// LS Electric XG5000 project: 래더
// PLC NewPLC
// module base 0 slot 0: 입출력 모듈:XBC-DR32H (DC 24V 입력, 릴레이 출력 32점)
// module base 0 slot 1: 위치결정 모듈:XBF-PD02A (위치결정 펄스(LD)출력형, 2축)
// module base 0 slot 2: 출력 모듈:XBE-TN/TP16A (트랜지스터 출력, 16점 (싱크출력/소스출력))

PROGRAM NewProgram (task: 스캔 프로그램)

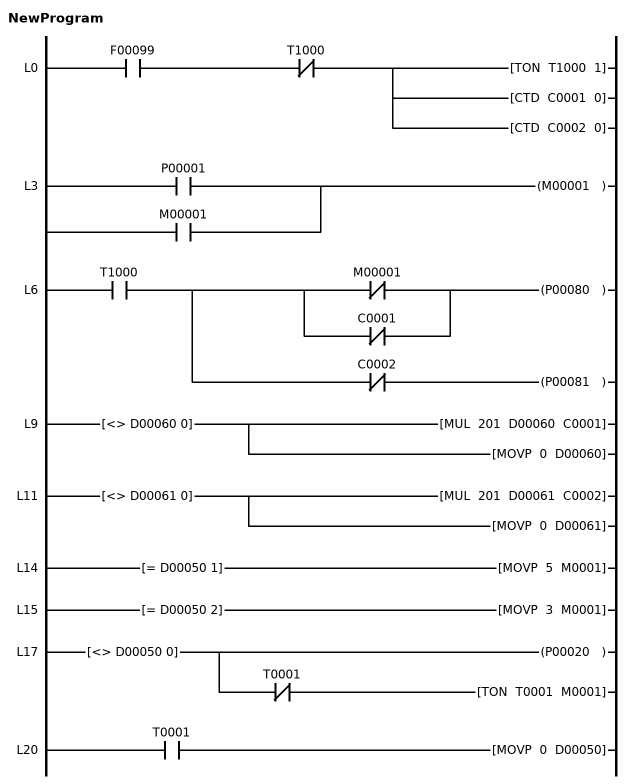
; L0
LOAD      F00099
AND NOT   T1000
TON       T1000 1
CTD       C0001 0
CTD       C0002 0
; L3
LOAD      P00001
OR        M00001
OUT       M00001
; L6
LOAD      T1000
MPUSH
LOAD NOT  M00001
OR NOT    C0001
AND LOAD
OUT       P00080
MPOP
AND NOT   C0002
OUT       P00081
; L9
LOAD<>    D00060 0
MUL       201 D00060 C0001
MOVP      0 D00060
; L11
LOAD<>    D00061 0
MUL       201 D00061 C0002
MOVP      0 D00061
; L14
LOAD=     D00050 1
MOVP      5 M0001
; L15
LOAD=     D00050 2
MOVP      3 M0001
; L17
LOAD<>    D00050 0
OUT       P00020
AND NOT   T0001
TON       T0001 M0001
; L20
LOAD      T0001
MOVP      0 D00050